FUNCTION_BLOCK SufficientFeedFlowBasic (* Basic Function Block Type *)
  (* Standard: 61499-2 *)
  (* Version 0.0, 9/23/2026, Schneider Electric, Template *)
  PACKAGE SE.Nereda;
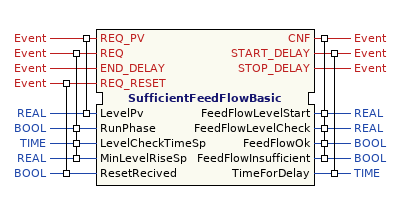
  EVENT_INPUT
    REQ_PV WITH LevelPv;
    REQ WITH LevelCheckTimeSp, MinLevelRiseSp, RunPhase; (* Normal Execution Request *)
    END_DELAY;
    REQ_RESET WITH ResetRecived;
  END_EVENT
  EVENT_OUTPUT
    CNF WITH FeedFlowLevelStart, FeedFlowOk, FeedFlowInsufficient, FeedFlowLevelCheck;
    START_DELAY WITH TimeForDelay;
    STOP_DELAY;
  END_EVENT
  VAR_INPUT
    LevelPv : REAL;
    RunPhase : BOOL;
    LevelCheckTimeSp : TIME;
    MinLevelRiseSp : REAL;
    ResetRecived : BOOL;
  END_VAR
  VAR_OUTPUT
    FeedFlowLevelStart : REAL;
    FeedFlowLevelCheck : REAL;
    FeedFlowOk : BOOL;
    FeedFlowInsufficient : BOOL;
    TimeForDelay : TIME;
  END_VAR
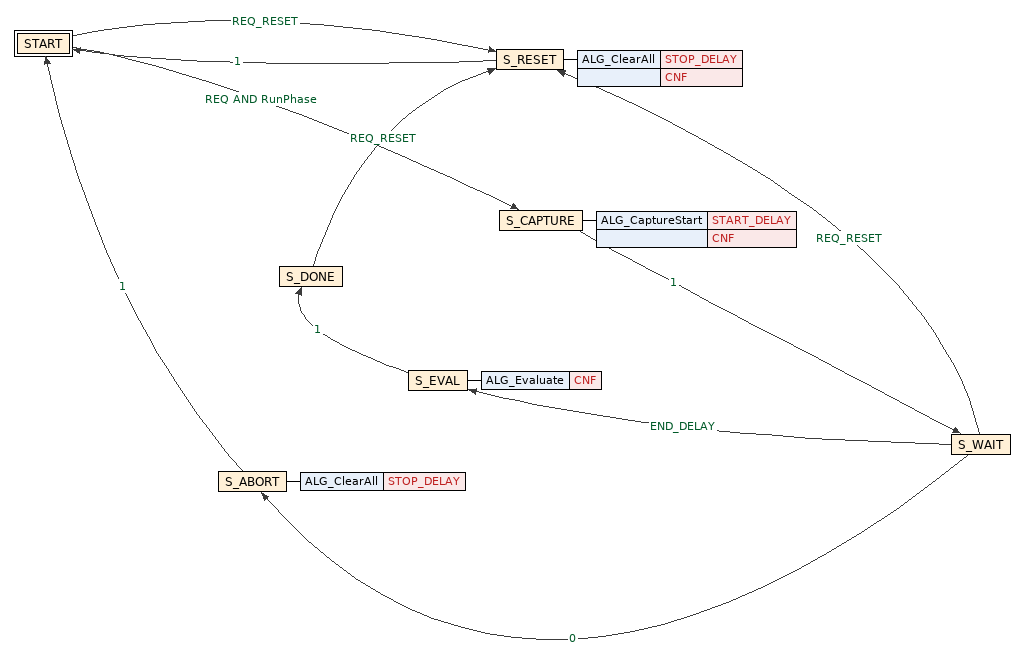
  EC_STATES
    START; (* Initial State *)
    S_CAPTURE : ALG_CaptureStart -> START_DELAY, -> CNF;
    S_WAIT;
    S_EVAL : ALG_Evaluate -> CNF;
    S_DONE;
    S_ABORT : ALG_ClearAll -> STOP_DELAY;
    S_RESET : ALG_ClearAll -> STOP_DELAY, -> CNF;
  END_STATES
  EC_TRANSITIONS
    START TO S_RESET := REQ_RESET;
    START TO S_CAPTURE := REQ AND RunPhase;
    S_CAPTURE TO S_WAIT := 1;
    S_WAIT TO S_RESET := REQ_RESET;
    S_WAIT TO S_ABORT := 0;
    S_WAIT TO S_EVAL := END_DELAY;
    S_EVAL TO S_DONE := 1;
    S_DONE TO S_RESET := REQ_RESET;
    S_ABORT TO START := 1;
    S_RESET TO START := 1;
  END_TRANSITIONS
  ALGORITHM ALG_CaptureStart IN ST:
FeedFlowLevelStart   := LevelPv;
FeedFlowLevelCheck   := 0.0;
FeedFlowOk           := FALSE;
FeedFlowInsufficient := FALSE;
TimeForDelay := LevelCheckTimeSp;
;
  END_ALGORITHM
  ALGORITHM ALG_Evaluate IN ST:
FeedFlowLevelCheck := LevelPv;
IF (FeedFlowLevelCheck - FeedFlowLevelStart) < MinLevelRiseSp THEN
    FeedFlowInsufficient := TRUE;
    FeedFlowOk           := FALSE;
ELSE
    FeedFlowOk           := TRUE;
    FeedFlowInsufficient := FALSE;
END_IF;
;
  END_ALGORITHM
  ALGORITHM ALG_ClearAll IN ST:
FeedFlowLevelStart   := 0.0;
FeedFlowLevelCheck   := 0.0;
FeedFlowOk           := FALSE;
FeedFlowInsufficient := FALSE;
;
  END_ALGORITHM
END_FUNCTION_BLOCK
